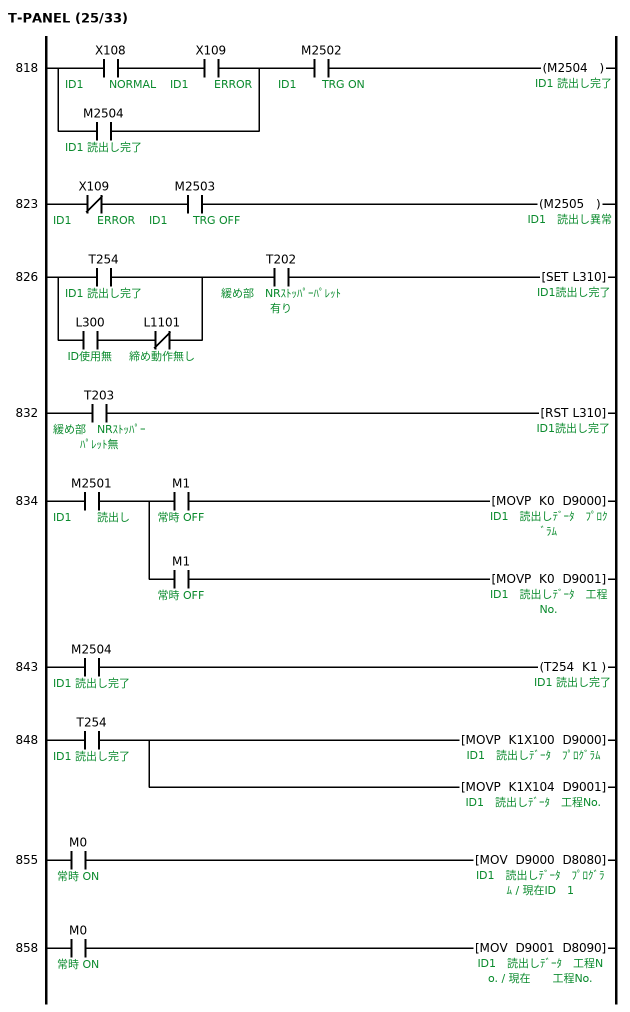
[picture p24: ladder of T-PANEL, rungs at steps 818 to 858]
818   LD      X108  ; ID1　　 NORMAL
      AND     X109  ; ID1　　 ERROR
      OR      M2504  ; ID1 読出し完了
      AND     M2502  ; ID1　 　TRG ON
      OUT     M2504  ; ID1 読出し完了
823   LDI     X109  ; ID1　　 ERROR
      AND     M2503  ; ID1　 　TRG OFF
      OUT     M2505  ; ID1　読出し異常
826   LD      T254  ; ID1 読出し完了
      LD      L300  ; ID使用無
      ANI     L1101  ; 締め動作無し
      ORB
      AND     T202  ; 緩め部　NRｽﾄｯﾊﾟｰﾊﾟﾚｯﾄ有り
      SET     L310  ; ID1読出し完了
832   LD      T203  ; 緩め部　NRｽﾄｯﾊﾟｰ ﾊﾟﾚｯﾄ無
      RST     L310  ; ID1読出し完了
834   LD      M2501  ; ID1　 　読出し
      MPS
      AND     M1  ; 常時 OFF
      MOVP    K0 D9000  ; ID1　読出しﾃﾞｰﾀ　ﾌﾟﾛｸﾞﾗﾑ
      MPP
      AND     M1  ; 常時 OFF
      MOVP    K0 D9001  ; ID1　読出しﾃﾞｰﾀ　工程No.
843   LD      M2504  ; ID1 読出し完了
      OUT     T254 K1  ; ID1 読出し完了
848   LD      T254  ; ID1 読出し完了
      MOVP    K1X100 D9000  ; ID1　　 READ DATA OD0
      MOVP    K1X104 D9001  ; ID1　　 READ DATA OD4
855   LD      M0  ; 常時 ON
      MOV     D9000 D8080
858   LD      M0  ; 常時 ON
      MOV     D9001 D8090  ; 現在　　工程No.
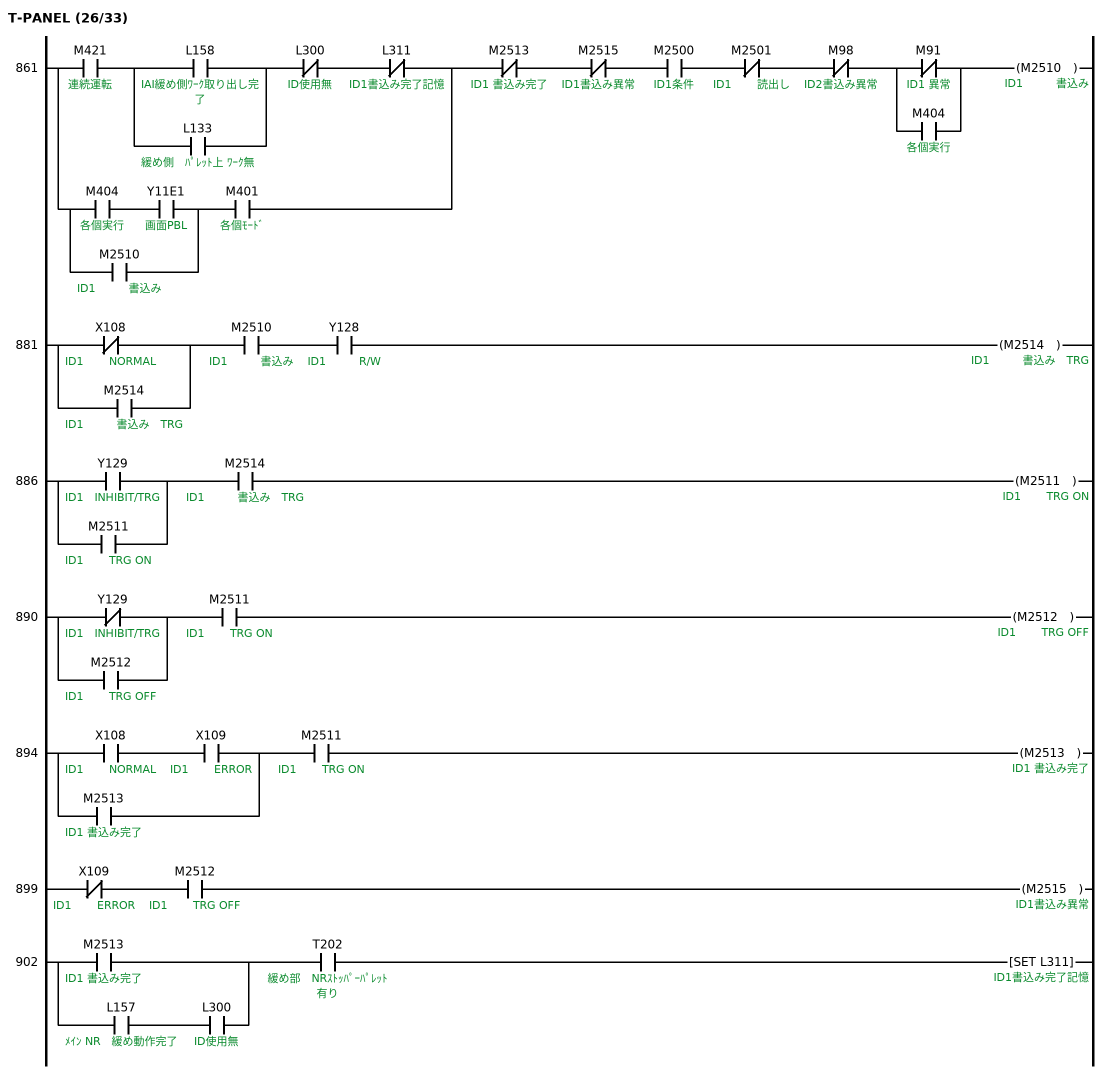
861   LD      M421  ; 連続運転
      LD      L158  ; IAI緩め側ﾜｰｸ取り出し完了
      OR      L133  ; 緩め側　ﾊﾟﾚｯﾄ上 ﾜｰｸ無
      ANB
      ANI     L300  ; ID使用無
      ANI     L311  ; ID1書込み完了記憶
      LD      M404  ; 各個実行
      AND     Y11E1  ; 画面PBL
      OR      M2510  ; ID1　　　書込み
      AND     M401  ; 各個ﾓｰﾄﾞ
      ORB
      ANI     M2513  ; ID1 書込み完了
      ANI     M2515  ; ID1書込み異常
      AND     M2500  ; ID1条件
      ANI     M2501  ; ID1　 　読出し
      ANI     M98  ; ID2書込み異常
      LDI     M91  ; ID1 異常
      OR      M404  ; 各個実行
      ANB
      OUT     M2510  ; ID1　　　書込み
881   LDI     X108  ; ID1　　 NORMAL
      OR      M2514  ; ID1　　　書込み　TRG
      AND     M2510  ; ID1　　　書込み
      AND     Y128  ; ID1　　　R/W
      OUT     M2514  ; ID1　　　書込み　TRG
886   LD      Y129  ; ID1　INHIBIT/TRG
      OR      M2511  ; ID1　 　TRG ON
      AND     M2514  ; ID1　　　書込み　TRG
      OUT     M2511  ; ID1　 　TRG ON
890   LDI     Y129  ; ID1　INHIBIT/TRG
      OR      M2512  ; ID1　 　TRG OFF
      AND     M2511  ; ID1　 　TRG ON
      OUT     M2512  ; ID1　 　TRG OFF
894   LD      X108  ; ID1　　 NORMAL
      AND     X109  ; ID1　　 ERROR
      OR      M2513  ; ID1 書込み完了
      AND     M2511  ; ID1　 　TRG ON
      OUT     M2513  ; ID1 書込み完了
899   LDI     X109  ; ID1　　 ERROR
      AND     M2512  ; ID1　 　TRG OFF
      OUT     M2515  ; ID1書込み異常
902   LD      M2513  ; ID1 書込み完了
      LD      L157  ; ﾒｲﾝ NR　緩め動作完了
      AND     L300  ; ID使用無
      ORB
      AND     T202  ; 緩め部　NRｽﾄｯﾊﾟｰﾊﾟﾚｯﾄ有り
      SET     L311  ; ID1書込み完了記憶
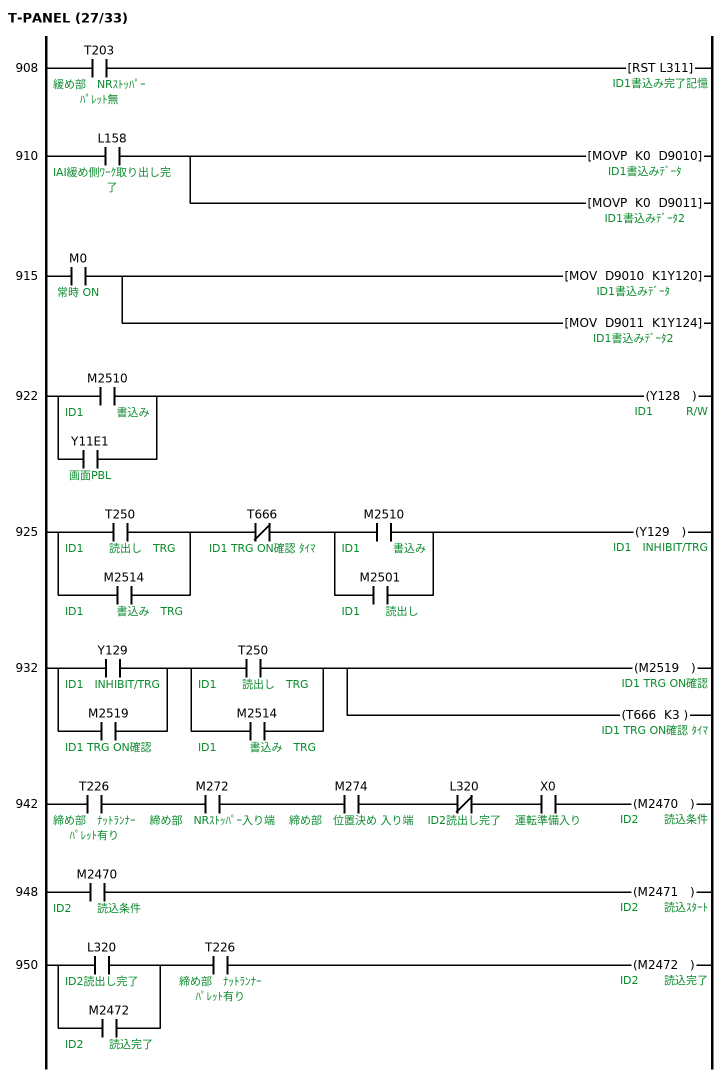
908   LD      T203  ; 緩め部　NRｽﾄｯﾊﾟｰ ﾊﾟﾚｯﾄ無
      RST     L311  ; ID1書込み完了記憶
910   LD      L158  ; IAI緩め側ﾜｰｸ取り出し完了
      MOVP    K0 D9010  ; ID1書込みﾃﾞｰﾀ
      MOVP    K0 D9011  ; ID1書込みﾃﾞｰﾀ2
915   LD      M0  ; 常時 ON
      MOV     D9010 K1Y120  ; ID1　　 WRITE DATA ID0
      MOV     D9011 K1Y124  ; ID1　WRITE DATA ID4
922   LD      M2510  ; ID1　　　書込み
      OR      Y11E1  ; 画面PBL
      OUT     Y128  ; ID1　　　R/W
925   LD      T250  ; ID1　 　読出し　TRG
      OR      M2514  ; ID1　　　書込み　TRG
      ANI     T666  ; ID1 TRG ON確認 ﾀｲﾏ
      LD      M2510  ; ID1　　　書込み
      OR      M2501  ; ID1　 　読出し
      ANB
      OUT     Y129  ; ID1　INHIBIT/TRG
932   LD      Y129  ; ID1　INHIBIT/TRG
      OR      M2519  ; ID1 TRG ON確認
      LD      T250  ; ID1　 　読出し　TRG
      OR      M2514  ; ID1　　　書込み　TRG
      ANB
      OUT     M2519  ; ID1 TRG ON確認
      OUT     T666 K3  ; ID1 TRG ON確認 ﾀｲﾏ
942   LD      T226  ; 締め部　ﾅｯﾄﾗﾝﾅｰ ﾊﾟﾚｯﾄ有り
      AND     M272  ; 締め部　NRｽﾄｯﾊﾟｰ入り端
      AND     M274  ; 締め部　位置決め 入り端
      ANI     L320  ; ID2読出し完了
      AND     X0  ; 運転準備入り
      OUT     M2470  ; ID2 　　読込条件
948   LD      M2470  ; ID2 　　読込条件
      OUT     M2471  ; ID2 　　読込ｽﾀｰﾄ
950   LD      L320  ; ID2読出し完了
      OR      M2472  ; ID2 　　読込完了
      AND     T226  ; 締め部　ﾅｯﾄﾗﾝﾅｰ ﾊﾟﾚｯﾄ有り
      OUT     M2472  ; ID2 　　読込完了
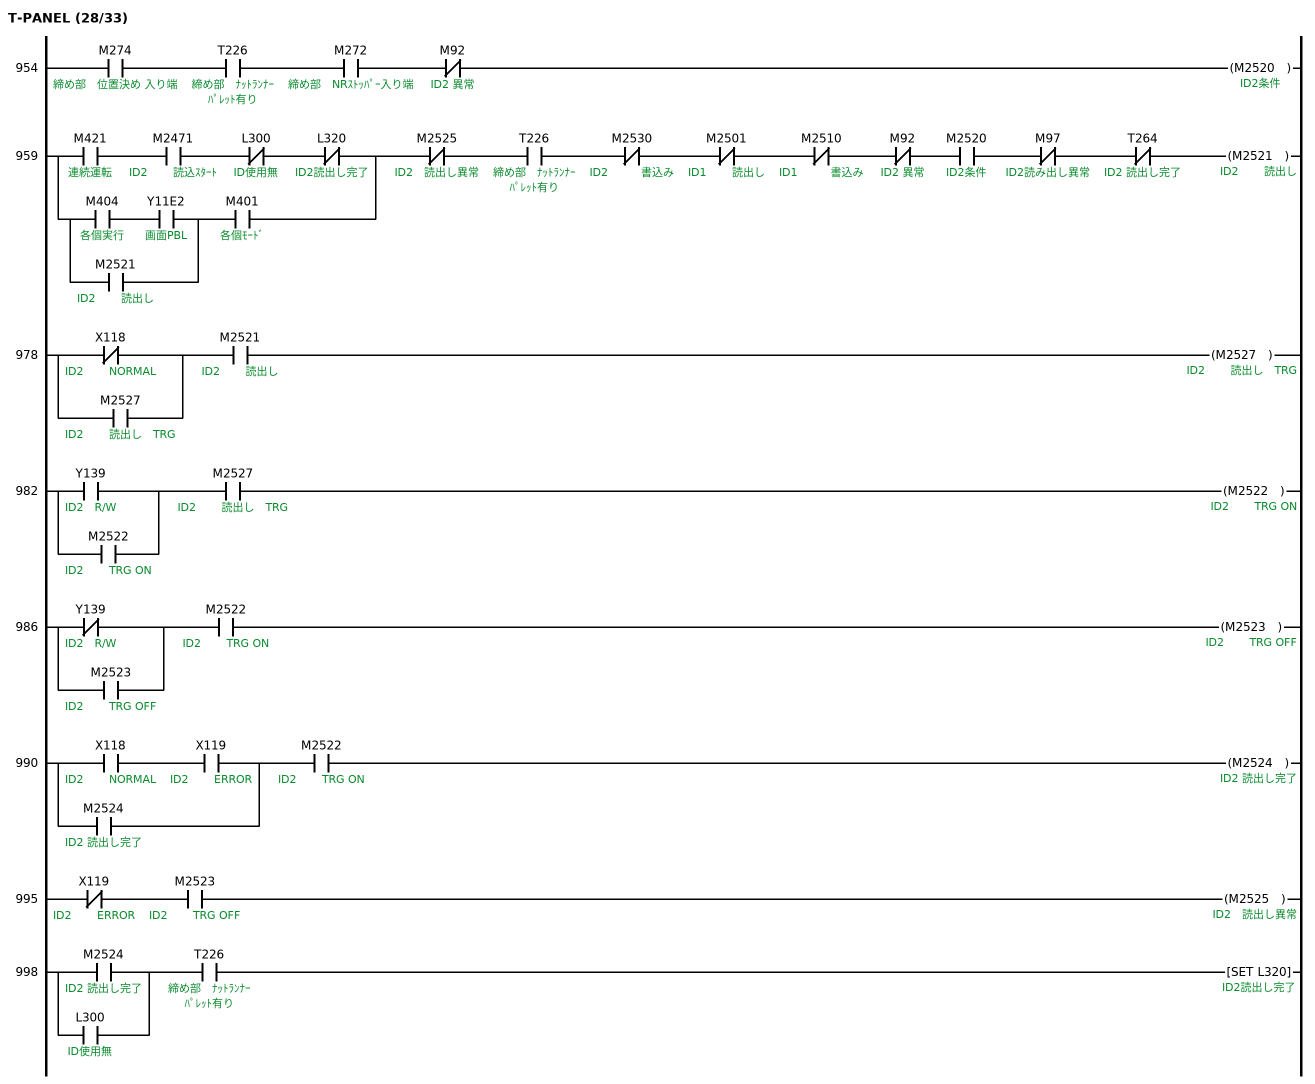
954   LD      M274  ; 締め部　位置決め 入り端
      AND     T226  ; 締め部　ﾅｯﾄﾗﾝﾅｰ ﾊﾟﾚｯﾄ有り
      AND     M272  ; 締め部　NRｽﾄｯﾊﾟｰ入り端
      ANI     M92  ; ID2 異常
      OUT     M2520  ; ID2条件
959   LD      M421  ; 連続運転
      AND     M2471  ; ID2 　　読込ｽﾀｰﾄ
      ANI     L300  ; ID使用無
      ANI     L320  ; ID2読出し完了
      LD      M404  ; 各個実行
      AND     Y11E2  ; 画面PBL
      OR      M2521  ; ID2　 　読出し
      AND     M401  ; 各個ﾓｰﾄﾞ
      ORB
      ANI     M2525  ; ID2　読出し異常
      AND     T226  ; 締め部　ﾅｯﾄﾗﾝﾅｰ ﾊﾟﾚｯﾄ有り
      ANI     M2530  ; ID2　　　書込み
      ANI     M2501  ; ID1　 　読出し
      ANI     M2510  ; ID1　　　書込み
      ANI     M92  ; ID2 異常
      AND     M2520  ; ID2条件
      ANI     M97  ; ID2読み出し異常
      ANI     T264  ; ID2 読出し完了
      OUT     M2521  ; ID2　 　読出し
978   LDI     X118  ; ID2　　 NORMAL
      OR      M2527  ; ID2　 　読出し　TRG
      AND     M2521  ; ID2　 　読出し
      OUT     M2527  ; ID2　 　読出し　TRG
982   LD      Y139  ; ID2　R/W
      OR      M2522  ; ID2　 　TRG ON
      AND     M2527  ; ID2　 　読出し　TRG
      OUT     M2522  ; ID2　 　TRG ON
986   LDI     Y139  ; ID2　R/W
      OR      M2523  ; ID2　 　TRG OFF
      AND     M2522  ; ID2　 　TRG ON
      OUT     M2523  ; ID2　 　TRG OFF
990   LD      X118  ; ID2　　 NORMAL
      AND     X119  ; ID2　　 ERROR
      OR      M2524  ; ID2 読出し完了
      AND     M2522  ; ID2　 　TRG ON
      OUT     M2524  ; ID2 読出し完了
995   LDI     X119  ; ID2　　 ERROR
      AND     M2523  ; ID2　 　TRG OFF
      OUT     M2525  ; ID2　読出し異常
998   LD      M2524  ; ID2 読出し完了
      OR      L300  ; ID使用無
      AND     T226  ; 締め部　ﾅｯﾄﾗﾝﾅｰ ﾊﾟﾚｯﾄ有り
      SET     L320  ; ID2読出し完了
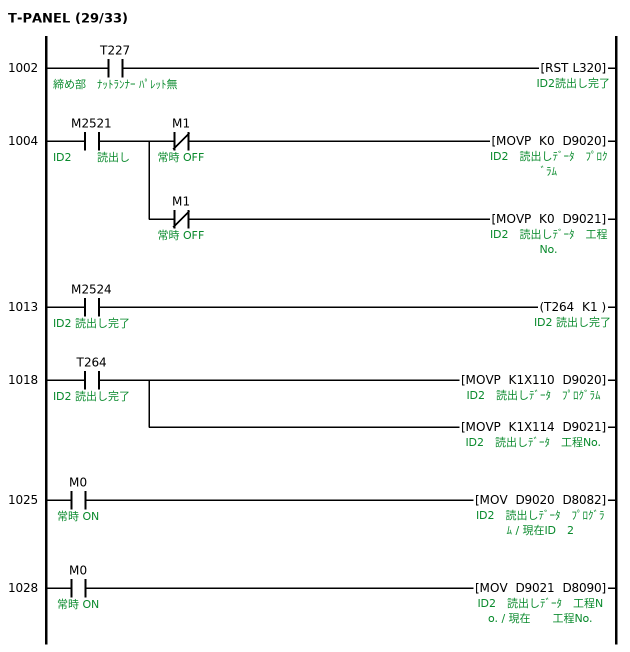
1002  LD      T227  ; 締め部　ﾅｯﾄﾗﾝﾅｰ ﾊﾟﾚｯﾄ無
      RST     L320  ; ID2読出し完了
1004  LD      M2521  ; ID2　 　読出し
      MPS
      ANI     M1  ; 常時 OFF
      MOVP    K0 D9020  ; ID2　読出しﾃﾞｰﾀ　ﾌﾟﾛｸﾞﾗﾑ
      MPP
      ANI     M1  ; 常時 OFF
      MOVP    K0 D9021  ; ID2　読出しﾃﾞｰﾀ　工程No.
1013  LD      M2524  ; ID2 読出し完了
      OUT     T264 K1  ; ID2 読出し完了
1018  LD      T264  ; ID2 読出し完了
      MOVP    K1X110 D9020  ; ID2　READ DATA OD0
      MOVP    K1X114 D9021  ; ID2　READ DATA OD4
1025  LD      M0  ; 常時 ON
      MOV     D9020 D8082  ; 現在ID　2
1028  LD      M0  ; 常時 ON
      MOV     D9021 D8090
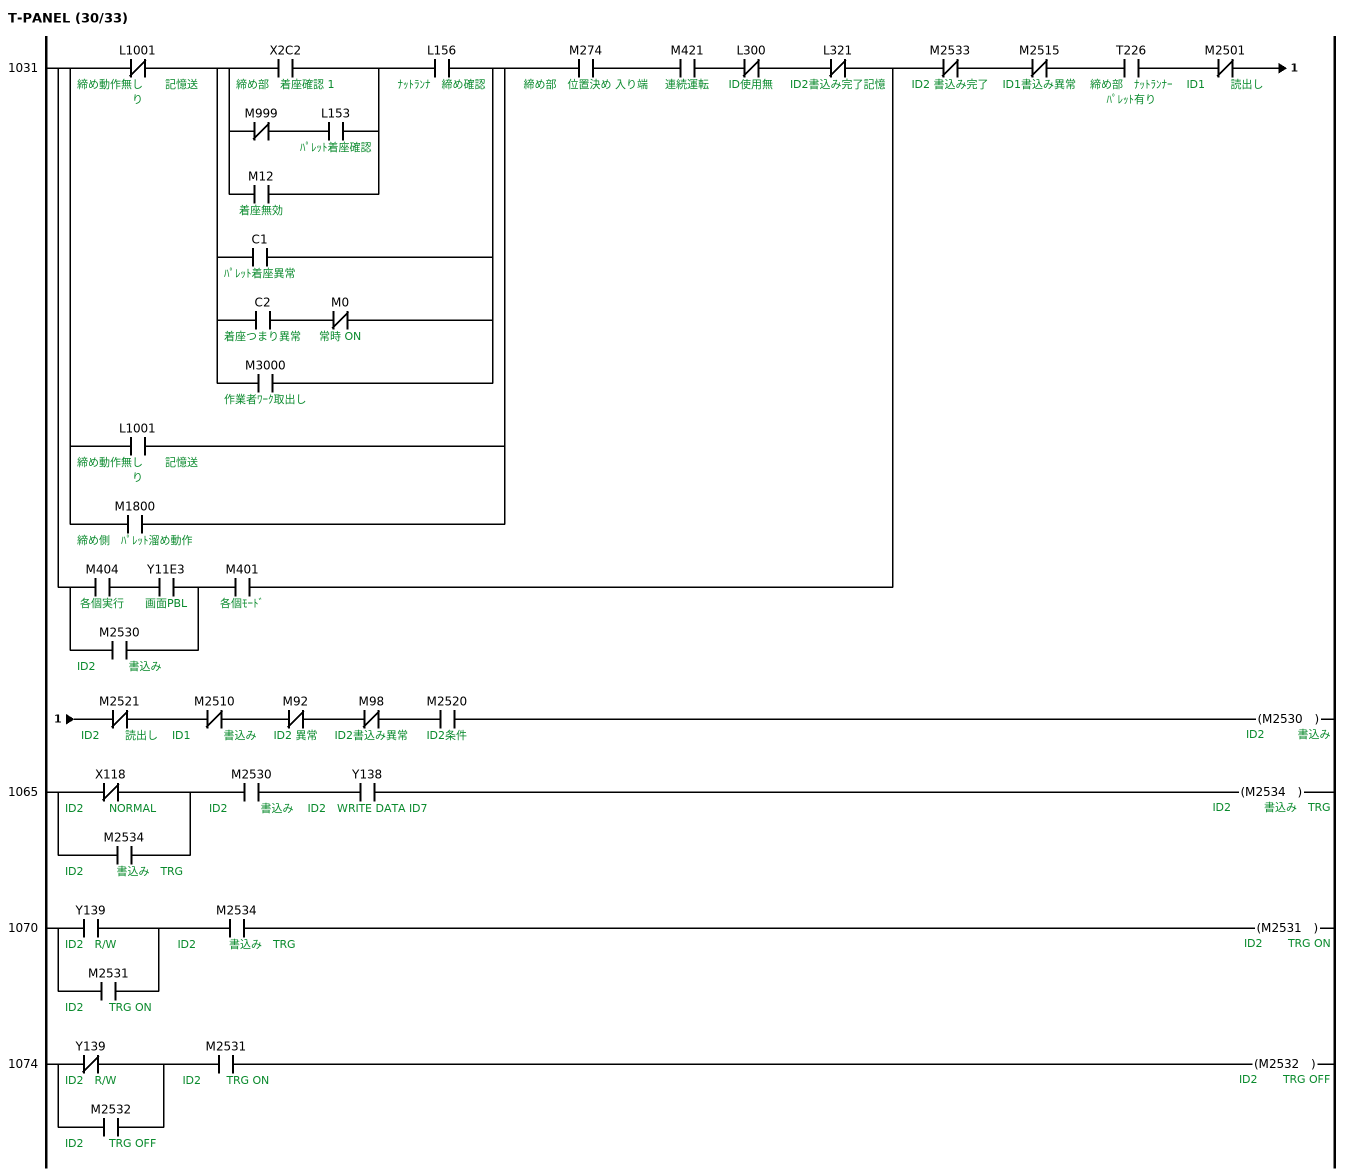
1031  LDI     L1001  ; 締め動作無し　　記憶送り
      LD      X2C2  ; 締め部　着座確認 1
      LDI     M999
      AND     L153  ; ﾊﾟﾚｯﾄ着座確認
      ORB
      OR      M12  ; 着座無効
      AND     L156  ; ﾅｯﾄﾗﾝﾅ　締め確認
      OR      C1  ; ﾊﾟﾚｯﾄ着座異常
      LD      C2  ; 着座つまり異常
      ANI     M0  ; 常時 ON
      ORB
      OR      M3000  ; 作業者ﾜｰｸ取出し
      ANB
      OR      L1001  ; 締め動作無し　　記憶送り
      OR      M1800  ; 締め側　ﾊﾟﾚｯﾄ溜め動作
      AND     M274  ; 締め部　位置決め 入り端
      AND     M421  ; 連続運転
      ANI     L300  ; ID使用無
      ANI     L321  ; ID2書込み完了記憶
      LD      M404  ; 各個実行
      AND     Y11E3  ; 画面PBL
      OR      M2530  ; ID2　　　書込み
      AND     M401  ; 各個ﾓｰﾄﾞ
      ORB
      ANI     M2533  ; ID2 書込み完了
      ANI     M2515  ; ID1書込み異常
      AND     T226  ; 締め部　ﾅｯﾄﾗﾝﾅｰ ﾊﾟﾚｯﾄ有り
      ANI     M2501  ; ID1　 　読出し
      ANI     M2521  ; ID2　 　読出し
      ANI     M2510  ; ID1　　　書込み
      ANI     M92  ; ID2 異常
      ANI     M98  ; ID2書込み異常
      AND     M2520  ; ID2条件
      OUT     M2530  ; ID2　　　書込み
1065  LDI     X118  ; ID2　　 NORMAL
      OR      M2534  ; ID2　　　書込み　TRG
      AND     M2530  ; ID2　　　書込み
      AND     Y138  ; ID2　WRITE DATA ID7
      OUT     M2534  ; ID2　　　書込み　TRG
1070  LD      Y139  ; ID2　R/W
      OR      M2531  ; ID2　 　TRG ON
      AND     M2534  ; ID2　　　書込み　TRG
      OUT     M2531  ; ID2　 　TRG ON
1074  LDI     Y139  ; ID2　R/W
      OR      M2532  ; ID2　 　TRG OFF
      AND     M2531  ; ID2　 　TRG ON
      OUT     M2532  ; ID2　 　TRG OFF
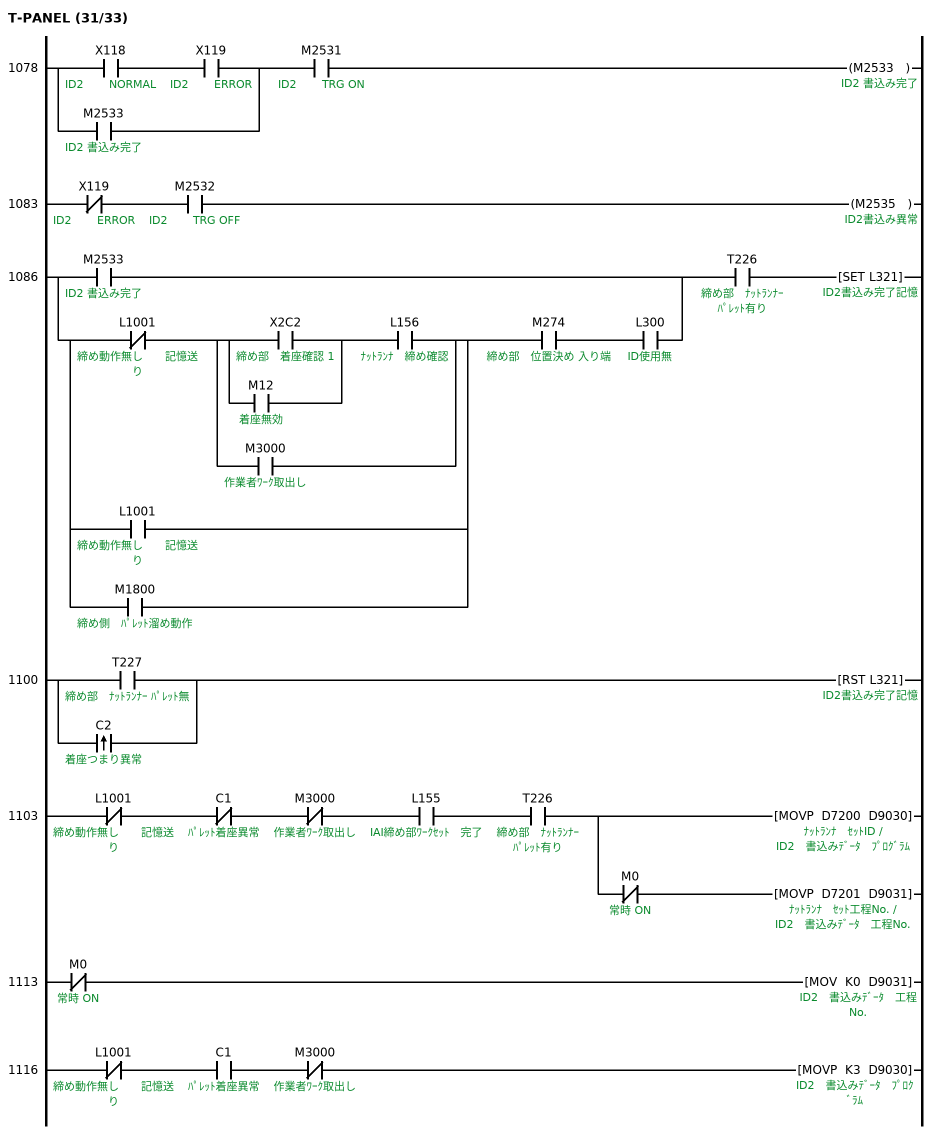
1078  LD      X118  ; ID2　　 NORMAL
      AND     X119  ; ID2　　 ERROR
      OR      M2533  ; ID2 書込み完了
      AND     M2531  ; ID2　 　TRG ON
      OUT     M2533  ; ID2 書込み完了
1083  LDI     X119  ; ID2　　 ERROR
      AND     M2532  ; ID2　 　TRG OFF
      OUT     M2535  ; ID2書込み異常
1086  LD      M2533  ; ID2 書込み完了
      LDI     L1001  ; 締め動作無し　　記憶送り
      LD      X2C2  ; 締め部　着座確認 1
      OR      M12  ; 着座無効
      AND     L156  ; ﾅｯﾄﾗﾝﾅ　締め確認
      OR      M3000  ; 作業者ﾜｰｸ取出し
      ANB
      OR      L1001  ; 締め動作無し　　記憶送り
      OR      M1800  ; 締め側　ﾊﾟﾚｯﾄ溜め動作
      AND     M274  ; 締め部　位置決め 入り端
      AND     L300  ; ID使用無
      ORB
      AND     T226  ; 締め部　ﾅｯﾄﾗﾝﾅｰ ﾊﾟﾚｯﾄ有り
      SET     L321  ; ID2書込み完了記憶
1100  LD      T227  ; 締め部　ﾅｯﾄﾗﾝﾅｰ ﾊﾟﾚｯﾄ無
      ORP     C2  ; 着座つまり異常
      RST     L321  ; ID2書込み完了記憶
1103  LDI     L1001  ; 締め動作無し　　記憶送り
      ANI     C1  ; ﾊﾟﾚｯﾄ着座異常
      ANI     M3000  ; 作業者ﾜｰｸ取出し
      AND     L155  ; IAI締め部ﾜｰｸｾｯﾄ　完了
      AND     T226  ; 締め部　ﾅｯﾄﾗﾝﾅｰ ﾊﾟﾚｯﾄ有り
      MOVP    D7200 D9030  ; ﾅｯﾄﾗﾝﾅ　ｾｯﾄID / ID2　書込みﾃﾞｰﾀ　ﾌﾟﾛｸﾞﾗﾑ
      ANI     M0  ; 常時 ON
      MOVP    D7201 D9031  ; ﾅｯﾄﾗﾝﾅ　ｾｯﾄ工程No. / ID2　書込みﾃﾞｰﾀ　工程No.
1113  LDI     M0  ; 常時 ON
      MOV     K0 D9031
1116  LDI     L1001  ; 締め動作無し　　記憶送り
      AND     C1  ; ﾊﾟﾚｯﾄ着座異常
      ANI     M3000  ; 作業者ﾜｰｸ取出し
      MOVP    K3 D9030
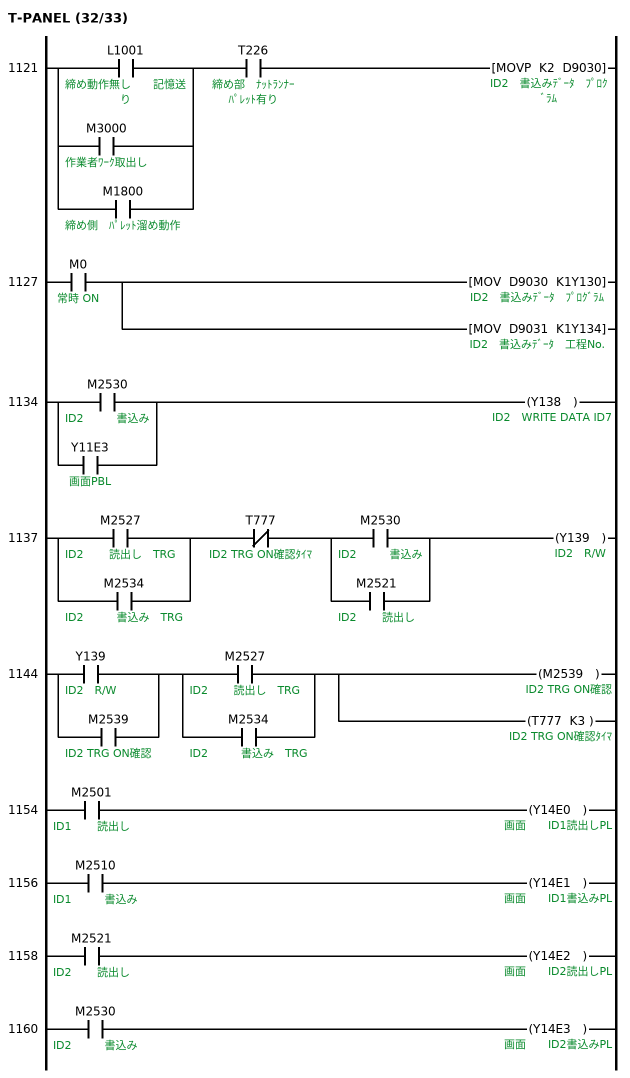
1121  LD      L1001  ; 締め動作無し　　記憶送り
      OR      M3000  ; 作業者ﾜｰｸ取出し
      OR      M1800  ; 締め側　ﾊﾟﾚｯﾄ溜め動作
      AND     T226  ; 締め部　ﾅｯﾄﾗﾝﾅｰ ﾊﾟﾚｯﾄ有り
      MOVP    K2 D9030
1127  LD      M0  ; 常時 ON
      MOV     D9030 K1Y130  ; ID2　INHIBIT/TRG
      MOV     D9031 K1Y134  ; ID2　WRITE DATA ID3
1134  LD      M2530  ; ID2　　　書込み
      OR      Y11E3  ; 画面PBL
      OUT     Y138  ; ID2　WRITE DATA ID7
1137  LD      M2527  ; ID2　 　読出し　TRG
      OR      M2534  ; ID2　　　書込み　TRG
      ANI     T777  ; ID2 TRG ON確認ﾀｲﾏ
      LD      M2530  ; ID2　　　書込み
      OR      M2521  ; ID2　 　読出し
      ANB
      OUT     Y139  ; ID2　R/W
1144  LD      Y139  ; ID2　R/W
      OR      M2539  ; ID2 TRG ON確認
      LD      M2527  ; ID2　 　読出し　TRG
      OR      M2534  ; ID2　　　書込み　TRG
      ANB
      OUT     M2539  ; ID2 TRG ON確認
      OUT     T777 K3  ; ID2 TRG ON確認ﾀｲﾏ
1154  LD      M2501  ; ID1　 　読出し
      OUT     Y14E0  ; 画面　　ID1読出しPL
1156  LD      M2510  ; ID1　　　書込み
      OUT     Y14E1  ; 画面　　ID1書込みPL
1158  LD      M2521  ; ID2　 　読出し
      OUT     Y14E2  ; 画面　　ID2読出しPL
1160  LD      M2530  ; ID2　　　書込み
      OUT     Y14E3  ; 画面　　ID2書込みPL
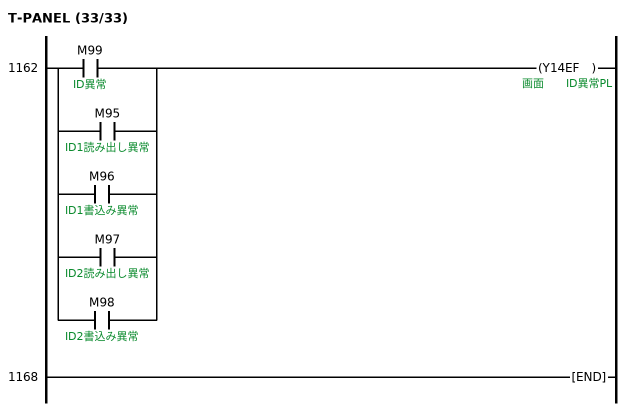
1162  LD      M99  ; ID異常
      OR      M95  ; ID1読み出し異常
      OR      M96  ; ID1書込み異常
      OR      M97  ; ID2読み出し異常
      OR      M98  ; ID2書込み異常
      OUT     Y14EF  ; 画面　　ID異常PL
1168  END
END_PROGRAM
